KUKA KRL data list: A28_screw_global.dat

&ACCESS RV
&COMMENT V_1_4_0
&PARAM DISKPATH = KRC:\R1\BMW_App
&REL 4
DEFDAT A28_screw_global PUBLIC
;********************************
;Date: 07.11.2018
;Programmer: AIUT
;Description: Global positions
;********************************


ENDDAT
